VAR_GLOBAL
	Eixo1 : AXIS_REF;
	Eixo2 : AXIS_REF;
END_VAR

(* stored: Version 1.1.0.1
   GVL Eixos: Id {530863fe-57e1-49d6-9324-1b69db309c3b} *)
